TYPE ST_AKM_Parameter :
STRUCT
	AutoQuittierung			: BOOL := 0;
	Temp_VL_blau_verfuegbar	: REAL;
	Temp_VL_gruen_verfuegbar: REAL;
	Temp_rot_soll_min		: REAL;
	Temp_rot_soll_max		: REAL;
	Temp_blau_soll_min		: REAL;
	Temp_gruen_soll_max		: REAL;
	Temp_gruen_soll_min		: REAL;
	Temp_blau_soll_max		: REAL;
END_STRUCT
END_TYPE

(* stored: Version 1.1.0.1, ProductVersion 3.1.4024.9
   DUT ST_AKM_Parameter: Id {8b432d57-46b5-4e3c-b077-f6d3203a1bb6} *)
